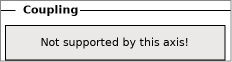
VISUALIZATION VISU_BaseAxis_Gearing  // 232x62
VAR_IN_OUT
	axis : BaseAxis;
    axisWidget : BaseAxisWidget;
END_VAR
    Button (141,25 80x35), "Decouple", input disabled if: axis.processes.gearOut.statuses.enabledStatus.disabled
        OnMouseClick: execute { axis.processes.gearOut.do_request := TRUE; }
    Frame (120,30 20x20)
        shows VISU_State_gray_orange(state := axisWidget.decoupled)
    Button (31,25 80x35), "Couple", input disabled if: axis.processes.gearIn.statuses.enabledStatus.disabled
        OnMouseClick: execute { axis.processes.gearIn.do_request := TRUE; }
    Frame (10,30 25x30)
        shows VISU_State_gray_green(state := axisWidget.coupled)
    Label (20,0 55x20), "Coupling"
    Line (80,10) (230,10)
    Line (0,10) (15,10)
    Rectangle (5,25 220x35), "Not supported by this axis!", invisible if: axis.isGearingSupported
END_VISUALIZATION

(* stored: Version 1.1.0.1, ProductVersion 3.1.4019.2
   Visu VISU_BaseAxis_Gearing: Id {f1e7b6d8-08f4-4a15-98da-20bacffb9d79} *)
